# B&R Automation Studio project SlidingGateDriveControl
Automation Studio 4.5.2.102

## Configuration SampleText

CPU 4PP065.0571-P74, AutomationRuntime D4.52, Build 4.1.2, Vc V4.25.0, Safety 1.6

### Task classes (Cpu.sw)
```
Cyclic#1 (cycle 2000 us, tolerance 0 us):
  ncsdcctrl <- ncsdcctrl.prg
Cyclic#4:
  Program <- Program.prg
DataObjects: Acp10sys
NcDataObjects: acp10etxen <- acp10etxen.dob, gAxis01a <- gAxis01obj.gAxis01a.dob, gAxis01i <- gAxis01obj.gAxis01i.dob
Binaries: ashwd, sysconf, asfw, arconfig, iomap, Acp10map, acp10cfg
Libraries: Acp10sdc, sys_lib, Runtime, asstring, Acp10man, Acp10par, NcGlobal, Acp10_MC, brsystem, AsBrStr, DriveLib, astime, fileio, powerlnk, asieccon
```

### Hardware
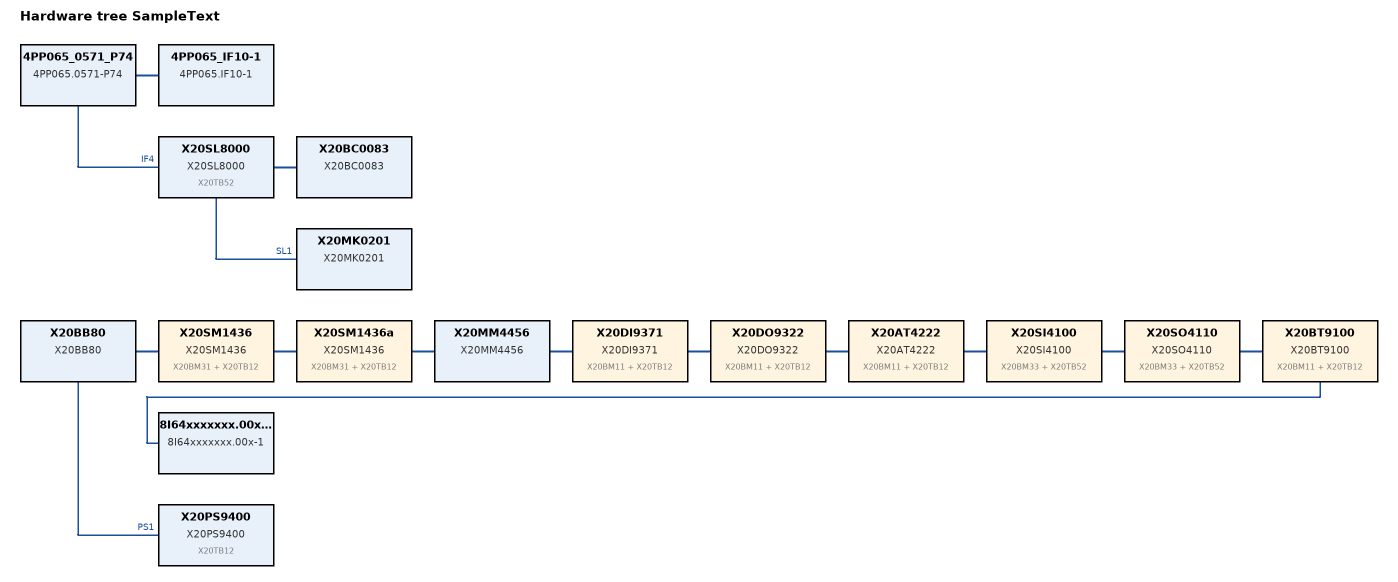
```
4PP065_0571_P74 : 4PP065.0571-P74 v1.1.2.0
  Connector IF4:
    EplInterfaceRedundant = 0
    EplEthInterfaceRedundant = 0
  Connector IF5:
    ActivateDevice = 1
    Mode = Manual
    InternetAddress = 10.0.1.13
    SubnetMask = 255.255.255.0
  ConfigurationID = labBR
  TimerDeviceType = EPLX2X
  TimerDevice = 4PP065_0571_P74.IF4
  TaskClassIdleTime = 2000
  Cyclic1Duration = 2000
  Cyclic1Tolerance = 0
  Cyclic1Output = 1
4PP065_IF10-1 : 4PP065.IF10-1 v1.0.3.0  [SS -> 4PP065_0571_P74.SS1]
8I64xxxxxxx.00x-1 : 8I64xxxxxxx.00x-1 v2.1.1.0  [X2X1 -> X20BT9100.X2X1 [Cable Type=X2XCable, Length=10, Version=1.0.0.2]]
  packedETAD = packed
  packedETI = packed
  packedCMDD = packed
  packedCMI = packed
  UNS = 220
  NCR = 10
  NSP = 890
  COS = 64
  RSC = 33000
X20AT4222 : X20AT4222 v1.2.3.0  [SS1 -> X20TB12e.SS; SL -> X20BM11c.SL1]
X20BB80 : X20BB80 v1.0.2.0
X20BC0083 : X20BC0083 v2.7.0.0  [PLK1 -> X20SL8000.PLK2 (NodeNumber=2) [Cable Type=PowerlinkCable, Length=10, Version=1.0.0.2]; SL -> X20BB80.SL1]
X20BM11 : X20BM11 v1.0.0.1  [X2X1 -> X20BM33a.X2X2]
X20BM11a : X20BM11 v1.0.0.1  [X2X1 -> X20MM4456.X2X2]
X20BM11b : X20BM11 v1.0.0.1  [X2X1 -> X20BM11a.X2X2]
X20BM11c : X20BM11 v1.0.0.1  [X2X1 -> X20BM11b.X2X2]
X20BM31 : X20BM31 v1.0.0.1  [X2X1 -> X20BB80.IF1]
X20BM31a : X20BM31 v1.0.0.1  [X2X1 -> X20BM31.X2X2]
X20BM33 : X20BM33 v1.0.0.4  [X2X1 -> X20BM11c.X2X2]
X20BM33a : X20BM33 v1.0.0.4  [X2X1 -> X20BM33.X2X2]
X20BT9100 : X20BT9100 v1.0.3.0  [SS1 -> X20TB12f.SS; SL -> X20BM11.SL1]
X20DI9371 : X20DI9371 v1.0.2.0  [SS1 -> X20TB12c.SS; SL -> X20BM11a.SL1]
X20DO9322 : X20DO9322 v1.0.3.0  [SS1 -> X20TB12d.SS; SL -> X20BM11b.SL1]
X20MK0201 : X20MK0201 v1.0.0.0  [SL -> X20SL8000.SL1]
X20MM4456 : X20MM4456 v1.1.5.0  [X2X1 -> X20BM31a.X2X2]
X20PS9400 : X20PS9400 v1.0.2.4  [SS1 -> X20TB12.SS; PS -> X20BB80.PS1]
X20SI4100 : X20SI4100 v1.10.1.1  [SS1 -> X20TB52.SS; SL -> X20BM33.SL1]
X20SL8000 : X20SL8000 v1.6.5.1  [PLK1 -> 4PP065_0571_P74.IF4 (NodeNumber=1) [Cable Type=PowerlinkCable, Length=10, Version=1.0.0.2]; PLK2 -> X20BC0083.PLK1 (NodeNumber=1) [Cable Type=PowerlinkCable, Length=10, Version=1.0.0.2]; SS1 -> X20TB52b.SS]
  SafeProject = SafeLOGIC-1
X20SM1436 : X20SM1436 v2.2.0.0  [SS1 -> X20TB12a.SS; SL -> X20BM31.SL1]
X20SM1436a : X20SM1436 v2.2.0.0  [SS1 -> X20TB12b.SS; SL -> X20BM31a.SL1]
X20SO4110 : X20SO4110 v1.10.1.1  [SS1 -> X20TB52a.SS; SL -> X20BM33a.SL1]
  SafeModuleID = 3
X20TB12 : X20TB12 v1.0.0.0
X20TB12a : X20TB12 v1.0.0.0
X20TB12b : X20TB12 v1.0.0.0
X20TB12c : X20TB12 v1.0.0.0
X20TB12d : X20TB12 v1.0.0.0
X20TB12e : X20TB12 v1.0.0.0
X20TB12f : X20TB12 v1.0.0.0
X20TB52 : X20TB52 v1.0.0.1
X20TB52a : X20TB52 v1.0.0.1
X20TB52b : X20TB52 v1.0.0.1
```

### IoMap.iom - 4PP065_0571_P74/IoMap.iom
```iecst
VAR_CONFIG
	Cyclic#1.gAxis01_DrvIf.iLifeCnt AT %IB."8I64xxxxxxx.00x-1".SDC_LifeCnt;
	Cyclic#1.gAxis01_DrvIf.oSetTime AT %QW."8I64xxxxxxx.00x-1".SDC_SetTime;
	Cyclic#1.::Program:driveSM.speed AT %QW."8I64xxxxxxx.00x-1".LFRD_Output;
	Cyclic#1.gAxis01_DiDoIf.iLifeCntDriveReady AT %IB."8I64xxxxxxx.00x-1".SDC_LifeCnt;
	Cyclic#1.gAxis01_DiDoIf.iLifeCntDriveEnable AT %IB."8I64xxxxxxx.00x-1".SDC_LifeCnt;
	Cyclic#1.gAxis01_ModuleOk AT %IX."8I64xxxxxxx.00x-1".ModuleOk;
	::Program:driveSM.state AT %IW."8I64xxxxxxx.00x-1".ETAD_Input;
	::Program:driveSM.command AT %QW."8I64xxxxxxx.00x-1".CMDD_Output;
	::Program:ledSM.led0 AT %QX."X20DO9322".DigitalOutput02;
	::Program:ledSM.led1 AT %QX."X20DO9322".DigitalOutput03;
	::Program:ledSM.led2 AT %QX."X20DO9322".DigitalOutput04;
	::Program:ledSM.led3 AT %QX."X20DO9322".DigitalOutput05;
	::Program:doorSM.direction AT %IX."X20DI9371".DigitalInput01;
	::Program:doorSM.sw0 AT %IX."X20DI9371".DigitalInput02;
	::Program:doorSM.sw1 AT %IX."X20DI9371".DigitalInput03;
	::Program:doorSM.sw2 AT %IX."X20DI9371".DigitalInput04;
	::Program:doorSM.sw3 AT %IX."X20DI9371".DigitalInput05;
END_VAR
```

### Acp10cfg.ncc - 4PP065_0571_P74/Motion/Acp10cfg.ncc
```
NcConfiguration (Version=3.16.0, NcSwId=Acp10)
  ACP10CF1_typ:
    cnt_nettrc_rec_drive = 1500
    bufsize_trace_upload = 1200
    tc_nc_man_task = Cyclic #1
    glob_pv_as_ncobject = Yes
    ncsys_dl_broadcast = Yes
    ncsys_dl_acp_reset = Yes
    safemc_log_err_to_ax = Yes
    network_init:
      ncsw_init_execute = Yes
      automatic_execute = No
      node_nr_warning = Yes
      net_err_before_ncact = Yes
    nettrc:
      enter_parsecrec = Yes
      enter_ncaction = Yes
      save_ring_startidx = Yes
    cam_prof_download:
      cam_dat_dl_parallel = No
      tc_cam_dl_parallel = Task class for NC Manager task
    sdc_if[0]:
      if_name = SDC_IF1
      mc_broadcast_size = 800
      mc_broadcast_extdat = No
```

## Configuration Simulation

### Hardware
```
PC_any : PC_any v1.1.0.0 (OrderNumber=PC)
```

## Logical view

Binary libraries used (declarations not repeated): Runtime, Operator, AsIecCon, astime, sys_lib, asstring, brsystem, AsBrStr, Acp10man, NcGlobal, Acp10par, Acp10sdc, Acp10_MC

### Data object Logical/acp10etxen (Ett)

- acp10etxen.ett (not shown)

- Data object Logical/gAxis01obj/gAxis01i (Ax) (no source held here)

### Library Logical/Libraries/DriveLib (ANSIC)

#### Types.typ - Exported data types
```iecst
TYPE
	ER_State :
		( (*Motor states*)
		ST_READY := 33, (*Ready to work*)
		ST_DISABLE := 64, (*Disable*)
		ST_SWITCHED_ON := 35 (*Switching states*)
		);
	ER_DoorState :
		( (*Door states*)
		ST_INIT, (*Initialization of parameters and waiting for switching on of the frequency converter*)
		ST_UNKNOWN, (*Gate in an unknown position*)
		ST_OPEN, (*The gate is open*)
		ST_CLOSE, (*The gate is close*)
		ST_ACC_POS, (*Gate acceleration towards opening*)
		ST_ACC_NEG, (*Gate acceleration towards closing*)
		ST_POS, (*Movement towards opening*)
		ST_NEG, (*Movement towards closing*)
		ST_DEC_POS, (*Slowdown of the gate towards the opening*)
		ST_DEC_NEG (*Slowdown of the gate towards the closing*)
		);
	ER_Command :
		( (*Motor commands*)
		CMD_SWITCH_ON := 7, (*Switching motor*)
		CMD_ENABLE := 15, (*Turning on the motor*)
		CMD_SHUTDOWN := 6, (*Motor shutdown*)
		CMD_DISABLE := 0 (*Motor disable*)
		);
END_TYPE
```

#### DriveLib.fun - Exported functions and function blocks
```iecst
FUNCTION_BLOCK FB_DriveSM (*This function block implements state switching for motor control*) (*$GROUP=User,$CAT=User,$GROUPICON=User.png,$CATICON=User.png*)
	VAR_INPUT
		state : UINT; (*Frequency converter status*)
		enable : BOOL; (*Function block operation signal*)
	END_VAR
	VAR_OUTPUT
		command : UINT; (*Frequency converter command*)
		speed : INT; (*Set speed*)
	END_VAR
END_FUNCTION_BLOCK

FUNCTION_BLOCK FB_LedSM (*This function block implements state switching to control indicators*) (*$GROUP=User,$CAT=User,$GROUPICON=User.png,$CATICON=User.png*)
	VAR_INPUT
		state : UINT; (*Gate condition*)
		led0 : BOOL; (*Function block operation signal*)
		led1 : BOOL; (*Function block operation signal*)
		led2 : BOOL; (*Function block operation signal*)
		led3 : BOOL; (*Function block operation signal*)
	END_VAR
	VAR_OUTPUT
		timer : INT; (*Set speed*)
	END_VAR
END_FUNCTION_BLOCK

FUNCTION_BLOCK FB_DoorSM (*This function block implements state switching for door control*) (*$GROUP=User,$CAT=User,$GROUPICON=User.png,$CATICON=User.png*)
	VAR_INPUT
		state : UINT; (*Gate condition*)
		sw0 : BOOL; (*Limit switch signal 1*)
		sw1 : BOOL; (*Limit switch signal 2*)
		sw2 : BOOL; (*Limit switch signal 3*)
		sw3 : BOOL; (*Limit switch signal 4*)
		direction : BOOL; (*Frequency converter command*)
	END_VAR
	VAR_OUTPUT
		speed : INT; (*Set speed*)
	END_VAR
END_FUNCTION_BLOCK
```

#### FB_DriveSM.c
```c
#include <bur/plctypes.h>
#ifdef __cplusplus
	extern "C"
	{
#endif
	#include "DriveLib.h"
#ifdef __cplusplus
	};
#endif
/* This function block implements state switching for motor control */
void FB_DriveSM(struct FB_DriveSM* inst)
{
	if(inst->enable == 0) inst->command = CMD_SHUTDOWN;
	else
	{
		switch(inst->state & 0x6F)
		{
			case ST_DISABLE:
				inst->command = CMD_SHUTDOWN;
				break;
			case ST_SWITCHED_ON:
				inst->command = CMD_SWITCH_ON;
				break;
			case ST_READY:
				inst->command = CMD_ENABLE;
				break;
		}
	}
}
```

#### FB_LedSM.c
```c
#include <bur/plctypes.h>
#ifdef __cplusplus
	extern "C"
	{
#endif
	#include "DriveLib.h"
#ifdef __cplusplus
	};
#endif
/* This function block implements state switching to control indicators */
void FB_LedSM(struct FB_LedSM* inst)
{
	switch(inst->state)
	{
		case ST_INIT:
			{
				break;
			}
		case ST_UNKNOWN:
			{
				if(inst->timer%10 == 9)
				{
					inst->led0 = !inst->led0;
					inst->led1 = !inst->led1;
					inst->led2 = !inst->led2;
					inst->led3 = !inst->led3;
				}
				break;
			}
		case ST_OPEN:
			{
				inst->led0 = 0;
				inst->led1 = 0;
				inst->led2 = 0;
				inst->led3 = 0;
				break;
			}
		case ST_CLOSE:
			{
				inst->led0 = 1;
				inst->led1 = 1;
				inst->led2 = 1;
				inst->led3 = 1;
				break;
			}
		case ST_ACC_POS:
			{
				if(inst->timer%10 == 4) inst->led0 = 1;
				inst->led1 = 0;
				inst->led2 = 0;
				inst->led3 = 0;
				break;
			}
		case ST_ACC_NEG:
			{
				inst->led0 = 1;
				inst->led1 = 1;
				inst->led2 = 1;
				if(inst->timer%10 == 4) inst->led3 = 0;
				break;
			}
		case ST_POS:
			{
				inst->led0 = 1;
				if(inst->timer%10 == 9) inst->led1 = 1;
				inst->led2 = 0;
				inst->led3 = 0;
				break;
			}
		case ST_NEG:
			{
				inst->led0 = 1;
				inst->led1 = 1;
				if(inst->timer%10 == 9) inst->led2 = 0;
				inst->led3 = 0;
				break;
			}
		case ST_DEC_POS:
			{
				inst->led0 = 1;
				inst->led1 = 1;
				if(inst->timer%10 == 4) inst->led2 = 1;
				inst->led3 = 0;
				break;
			}
		case ST_DEC_NEG:
			{
				inst->led0 = 1;
				if(inst->timer%10 == 4) inst->led1 = 0;
				inst->led2 = 0;
				inst->led3 = 0;
				break;
			}
	}
}
```

#### FB_DoorSM.c
```c
#include <bur/plctypes.h>
#ifdef __cplusplus
	extern "C"
	{
#endif
	#include "DriveLib.h"
#ifdef __cplusplus
	};
#endif
/* This function block implements state switching for door control */
void FB_DoorSM(struct FB_DoorSM* inst)
{
	switch(inst->state)
	{
		case ST_INIT:
			{
				if(inst->sw0 == 0 && inst->sw1 == 0 && inst->sw2 == 0 && inst->sw3 == 0) inst->state = ST_UNKNOWN;
				break;
			}
		case ST_UNKNOWN:
			{
				if(inst->direction == 0 && inst->sw0 == 1) inst->state = ST_OPEN;
				if(inst->direction == 1 && inst->sw3 == 1) inst->state = ST_CLOSE;
				break;
			}
		case ST_OPEN:
			{
				inst->speed = 0;
				if(inst->direction == 0) inst->state = ST_ACC_POS;
				break;
			}
		case ST_CLOSE:
			{
				inst->speed = 0;
				if(inst->direction == 1) inst->state = ST_ACC_NEG;
				break;
			}
		case ST_ACC_POS:
			{
				inst->speed = 200;
				if(inst->sw1 == 1) inst->state = ST_POS;
				if(inst->direction == 1) inst->state = ST_DEC_NEG;
				break;
			}
		case ST_ACC_NEG:
			{
				inst->speed = -200;
				if(inst->sw2 == 1) inst->state = ST_NEG;
				if(inst->direction == 0) inst->state = ST_DEC_POS;
				break;
			}
		case ST_POS:
			{
				inst->speed = 400;
				if(inst->sw2 == 1) inst->state = ST_DEC_POS;
				if(inst->direction == 1) inst->state = ST_NEG;
				break;
			}
		case ST_NEG:
			{
				inst->speed = -400;
				if(inst->sw1 == 1) inst->state = ST_DEC_NEG;
				if(inst->direction == 0) inst->state = ST_POS;
				break;
			}
		case ST_DEC_POS:
			{
				inst->speed = 100;
				if(inst->sw3 == 1) inst->state = ST_CLOSE;
				break;
			}
		case ST_DEC_NEG:
			{
				inst->speed = -100;
				if(inst->sw0 == 1) inst->state = ST_OPEN;
				break;
			}
	}
}
```

### Program Logical/Program

#### Variables.var
```iecst
VAR
	driveSM : FB_DriveSM := (0); (*Variable motor control*)
	doorSM : FB_DoorSM := (0); (*Gate control variable*)
	ledSM : FB_LedSM := (0); (*Indicator control variable*)
END_VAR
```

#### Main.c
```c
#include <bur/plctypes.h>

#ifdef _DEFAULT_INCLUDES
	#include <AsDefault.h>
#endif

void _INIT ProgramInit(void)
{
	driveSM.enable = 1;
}

void _CYCLIC ProgramCyclic(void)
{
	FB_DoorSM(&doorSM);

	driveSM.speed = doorSM.speed;
	FB_DriveSM(&driveSM);

	ledSM.state = doorSM.state;
	FB_LedSM(&ledSM);
	ledSM.timer++;
}

void _EXIT ProgramExit(void)
{

}
```

Listed in the project but not available here: Logical/gAxis01obj/gAxis01a, Logical/Libraries/DriveLib/Constants.var
